// TIA Portal V16 export
// export: Created 2021-06-29T09:40:51.540039Z, ExportSetting WithDefaults, WithReadOnly, DisplayName Totally Integrated Automation Portal, DisplayVersion V16 Update 3, DisplayName TIA Portal Version Control Interface, DisplayVersion V16 Update 2, DisplayName TIA Portal Openness, DisplayVersion V16 Update 3, DisplayName SINAMICS Startdrive Advanced, DisplayVersion V16, DisplayName SINAMICS Startdrive G130, G150, S120, S150, SINAMICS MV, S210, DisplayVersion V16, DisplayName SINAMICS Startdrive G110M, G120, G120C, G120D, G120P, DisplayVersion V16, DisplayName STEP 7 Professional, DisplayVersion V16 Update 3, DisplayName SIMATIC Energy Suite, DisplayVersion V16, DisplayName STEP 7 Safety, DisplayVersion V16, DisplayName WinCC Advanced, DisplayVersion V16 Update 3
Screen "interruttore"  1366x768, Number=2
  ScreenLayer 
    Group "Group"
      Rectangle "Rettangolo_1" at 44,30 size 138x117
      Circle "Cerchio_1" at 58,60 size 34x34
        RangeAppearanceAnimation "RangeAppearanceAnimation"
          tag BSA01_STATO
          0..0: back #ff0000, fore #181c31
          1..1: back #00ff00, fore #181c31
      TextField "Casella di testo_1" at 58,30 size 60x25  Text="Titolo"
      TextField "Casella di testo_2" at 98,63 size 56x25  Text="Stato"
      TextField "Casella di testo_3" at 98,109 size 80x25  Text="Termico"
      Circle "Cerchio_2" at 58,102 size 34x34
        RangeAppearanceAnimation "RangeAppearanceAnimation"
          tag BSA01_TERMICO
          0..0: back #ff0000, fore #181c31
          1..1: back #00ff00, fore #181c31
